{attribute 'qualified_only'}
VAR_GLOBAL
  //---------------------------------------------------------------------------
  // XTS Station
  //  - handshakes mover in station with extern control
  //  - station parameters (positions, gap, dyn. constraints, description...)
  StationStart        : ST_STATION_PARAMETER;   // Xts transport is sending all mover to this position (CMD_TRANSPORT_START)



  //---------------------------------------------------------------------------
  // XTS
  // XTS TransportUnit
  //  - handles request for XPU, Group, Mover, StartUp, ReStart
  XtsTransport        : fb_TransportUnit;

  XtsTransportCtrl    : ST_XTS_TRANSPORT_CTRL;
  XtsTransportState   : ST_XTS_TRANSPORT_STATE;


  //---------------------------------------------------------------------------
  // XPU
  // XTS-Utility checks
  Xpu             : fb_XpuCtrl;

  XpuCtrl         : ST_XPU_CTRL;
  XpuState        : ST_XPU_STATE;
  XpuInfo         : ST_XPU_INFO;
  XpuModules      : ARRAY[1..MAX_MODULE] OF Tc3_XTS_Utility.ST_InfoDataView;


  //---------------------------------------------------------------------------
  // Collision avoidance group CA
  //
  // - add mover to group
  // - build group
  // - clear group
  CaGroup         : FB_CaGroup;
  CaGroupItf      : I_XtsTransport_CaGroup;

  // cyclic mapping to MOTION/Objects/CaGroup 
  CaGroupRef      : Tc3_McCoordinatedMotion.AXES_GROUP_REF;

  // Info data from CaGroup FB
  CaGroupInfo     : ST_GROUP_INFO;
  //---------------------------------------------------------------------------

  //---------------------------------------------------------------------------
  // MC2 encapsulation, CA movement
  Mover           : ARRAY[1..MAX_MOVER] OF fb_Mover;
  MoverItf        : ARRAY[1..MAX_MOVER] OF I_XtsTransport_Mover;

  LastPosition    : ARRAY[1..MAX_MOVER] OF LREAL;
  LastGap         : ARRAY[1..MAX_MOVER] OF LREAL;

  MoverInfo       : ARRAY[1..MAX_MOVER] OF ST_MOVER_INFO;

  MoveData        : ARRAY[1..MAX_MOVER] OF ST_MOVE_DATA;
  GearData        : ARRAY[1..MAX_MOVER] OF ST_GEAR_DATA;
  
  // cyclic mapping to MOTION/Axes
  AxisRefMover    : ARRAY[1..MAX_MOVER] OF Tc2_MC2.AXIS_REF;
  //---------------------------------------------------------------------------
END_VAR

(* stored: Version 1.1.0.1, ProductVersion 3.1.4024.12
   GVL GVL_XTS: Id {4ca68d43-ee83-480c-9a51-2e5c312f57c1} *)
